// TIA Portal V18 export
TYPE "UDT_Motion_Point_V90"
   STRUCT
      Pos : DInt;   // Target Position (mm/deg)
      Vel : Int;   // Target Velocity (mm/s or rpm)
   END_STRUCT;
END_TYPE
